(* CoDeSys 2.3.9.59 project: PD4.pro *)
(* Libraries: Standard.lib, SYSLIBCALLBACK.LIB *)

(* PLC configuration (modules and I/O channels)
Configuration EC4P-200 [Root] node -1, in %IB0 out %QB0 {EC4P_RestartPwrOn = WARMSTART; EC4P_MaxCycleTime = 20; EC4P_Com1BaudRate = 38400; EC4P_CAN1BaudRate = 125KBaud; EC4P_RoutingId = 127; EC4P_EasyNetId = 1; EC4P_EasyNetCfg = 0; EC4P_EasyNetCycleTime = 50; EC4P_RoutingChannel = CAN1; EC4P_IPFlags = 0; EC4P_IPAddress = 0; EC4P_SubNetMask = 0; EC4P_DefaultGateway = 0; EC4P_SummerWinterFlags = 0; EC4P_SummerWinterRule1 = 0; EC4P_SummerWinterRule2 = 0}
  Local I/O [EC4P_LocalIO] node 0, in %IB0 out %QB0 {EC4P_LocalInt = 0}
    I1 AT %IX0.0 [LocalBitInput] Input I1
    I2 AT %IX0.1 [LocalBitInput] Input I2
    I3 AT %IX0.2 [LocalBitInput] Input I3
    I4 AT %IX0.3 [LocalBitInput] Input I4
    I5 AT %IX0.4 [LocalBitInput] Input I5
    I6 AT %IX0.5 [LocalBitInput] Input I6
    I7 AT %IX0.6 [LocalBitInput] Input I7
    I8 AT %IX0.7 [LocalBitInput] Input I8
    I9 AT %IX1.0 [LocalBitInput] Input I9
    I10 AT %IX1.1 [LocalBitInput] Input I10
    I11 AT %IX1.2 [LocalBitInput] Input I11
    I12 AT %IX1.3 [LocalBitInput] Input I12
    I13 AT %IX1.4 [LocalDiagInput] Diagnostic Input I13
    I14 AT %IX1.5 [LocalDiagInput] Diagnostic Input I14
    I15 AT %IX1.6 [LocalDiagInput] Diagnostic Input I15
    I16 AT %IX1.7 [LocalDiagInput] Diagnostic Input I16
    I7_Analog AT %IW2 [LocalAnalogIn] Input I7, 10Bit, 0-10VDC
    I8_Analog AT %IW4 [LocalAnalogIn] Input I8, 10Bit, 0-10VDC
    I11_Analog AT %IW6 [LocalAnalogIn] Input I11, 10Bit, 0-10VDC
    I12_Analog AT %IW8 [LocalAnalogIn] Input I12, 10Bit, 0-10VDC
    Transistor Outputs [EC4P_TOutputs] node 0, in %IB10 out %QB0
      Q1 AT %QX0.0 [LocalBitOutput] Transistor-Output Q1
      Q2 AT %QX0.1 [LocalBitOutput] Transistor-Output Q2
      Q3 AT %QX0.2 [LocalBitOutput] Transistor-Output Q3
      Q4 AT %QX0.3 [LocalBitOutput] Transistor-Output Q4
      Q5 AT %QX0.4 [LocalBitOutput] Transistor-Output Q5
      Q6 AT %QX0.5 [LocalBitOutput] Transistor-Output Q6
      Q7 AT %QX0.6 [LocalBitOutput] Transistor-Output Q7
      Q8 AT %QX0.7 [LocalBitOutput] Transistor-Output Q8
    No Analog Output [EC4P_NoAnalogOutput] node 1, in %IB10 out %QB1
    No Keys [EC4P_NoKeys] node 2, in %IB10 out %QB1
    No Counter [EC4P_NoCounter] node 3, in %IB10 out %QB1
  Extension [EC4P_Extension] node 1, in %IB10 out %QB1
    No Extension [EC4P_NoExtension] node 0, in %IB10 out %QB1
*)

(* POU PLC_PRG, FBD *)
PROGRAM PLC_PRG
VAR
	sum: input_sum;
	segment: segment_driver;
END_VAR
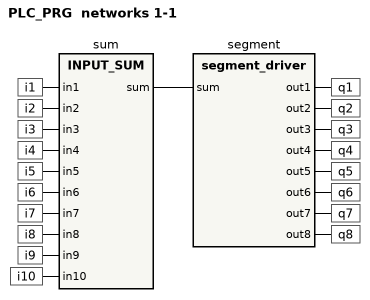
_FBD_ (* Function Block Diagram *)
NETWORK 1
	segment:segment_driver(sum: sum:INPUT_SUM(in1: i1, in2: i2, in3: i3, in4: i4, in5: i5, in6: i6, in7: i7, in8: i8, in9: i9, in10: i10), out2 => q2, out3 => q3, out4 => q4, out5 => q5, out6 => q6, out7 => q7, out8 => q8) => q1
_END_FBD_
(* the same logic as Structured Text *)
(* Network 1 *)
sum(in1 := i1, in2 := i2, in3 := i3, in4 := i4, in5 := i5, in6 := i6, in7 := i7, in8 := i8, in9 := i9, in10 := i10);
segment(sum := sum.sum);
q2 := segment.out2;
q3 := segment.out3;
q4 := segment.out4;
q5 := segment.out5;
q6 := segment.out6;
q7 := segment.out7;
q8 := segment.out8;
q1 := segment.out1;
END_PROGRAM

(* POU input_sum, ST *)
FUNCTION_BLOCK input_sum
VAR_INPUT
	in1, in2, in3, in4, in5, in6, in7, in8, in9, in10: BOOL;
END_VAR
VAR_OUTPUT
	sum: WORD;
END_VAR
VAR
END_VAR
sum := BOOL_TO_INT(in1) + BOOL_TO_INT(in2) + BOOL_TO_INT(in3) + BOOL_TO_INT(in4) + BOOL_TO_INT(in5) + BOOL_TO_INT(in6)+ BOOL_TO_INT(in7) + BOOL_TO_INT(in8) + BOOL_TO_INT(in9) + BOOL_TO_INT(in10);
END_FUNCTION_BLOCK

(* POU segment_driver, ST *)
FUNCTION_BLOCK segment_driver
VAR_INPUT
	sum: WORD;
END_VAR
VAR_OUTPUT
	out1, out2, out3, out4, out5, out6, out7, out8: BOOL;
END_VAR
VAR
END_VAR
CASE sum OF
0:
	out1 := 0;
	out2 := 0;
	out3 := 0;
	out4 := 0;
	out5 := 0;
	out6 := 0;
	out7 := 0;
	out8 := 1;
1:
	out1 := 0;
	out2 := 1;
	out3 := 0;
	out4 := 1;
	out5 := 1;
	out6 := 1;
	out7 := 1;
	out8 := 0;
2:
	out1 := 0;
	out2 := 0;
	out3 := 0;
	out4 := 1;
	out5 := 1;
	out6 := 0;
	out7 := 0;
	out8 := 0;
3:
	out1 := 1 ;
	out2 := 0;
	out3 := 1;
	out4 := 1;
	out5 := 1;
	out6 := 0;
	out7 := 1;
	out8 := 0;
4:
	out1 := 1;
	out2 := 1;
	out3 := 0;
	out4 := 1;
	out5 := 1;
	out6 := 0;
	out7 := 1;
	out8 := 0;
5:
	out1 := 1;
	out2 := 0;
	out3 := 1;
	out4 := 1;
	out5 := 1;
	out6 := 0;
	out7 := 1;
	out8 := 0;
6:
	out1 := 0;
	out2 := 1;
	out3 := 0;
	out4 := 0;
	out5 := 1;
	out6 := 0;
	out7 := 0;
	out8 := 0;
7:
	out1 := 0;
	out2 := 0;
	out3 := 0;
	out4 := 1;
	out5 := 1;
	out6 := 1;
	out7 := 0;
	out8 := 0;
8:
	out1 := 1;
	out2 := 1;
	out3 := 0;
	out4 := 1;
	out5 := 0;
	out6 := 1;
	out7 := 1;
	out8 := 0;
9:
	out1 := 1;
	out2 := 1;
	out3 := 0;
	out4 := 1;
	out5 := 1;
	out6 := 1;
	out7 := 0;
	out8 := 0;
10:
	out1 := 1;
	out2 := 1;
	out3 := 1;
	out4 := 1;
	out5 := 1;
	out6 := 1;
	out7 := 0;
	out8 := 0;
ELSE
	out1 := 0;
	out2 := 0;
	out3 := 0;
	out4 := 0;
	out5 := 0;
	out6 := 0;
	out7 := 0;
	out8 := 0;
END_CASE;
END_FUNCTION_BLOCK

(* Visualisation gui
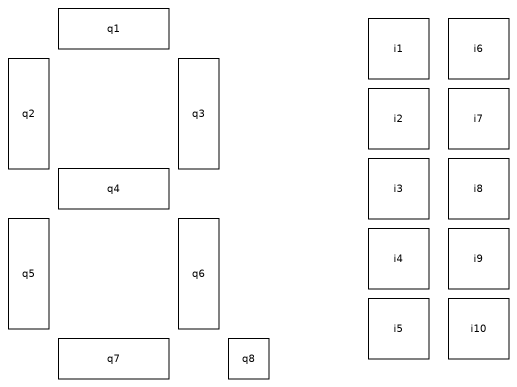
rectangle at (400,50)-(461,111): text "i1"; alarm colour if i1; toggles i1
rectangle at (400,120)-(461,181): text "i2"; alarm colour if i2; toggles i2
rectangle at (400,190)-(461,251): text "i3"; alarm colour if i3; toggles i3
rectangle at (480,50)-(541,111): text "i6"; alarm colour if i6; toggles i6
rectangle at (480,120)-(541,181): text "i7"; alarm colour if i7; toggles i7
rectangle at (480,190)-(541,251): text "i8"; alarm colour if i8; toggles i8
rectangle at (400,260)-(461,321): text "i4"; alarm colour if i4; toggles i4
rectangle at (400,330)-(461,391): text "i5"; alarm colour if i5; toggles i5
rectangle at (480,260)-(541,321): text "i9"; alarm colour if i9; toggles i9
rectangle at (480,330)-(541,391): text "i10"; alarm colour if i10; toggles i10
rectangle at (90,40)-(201,81): text "q1"; alarm colour if q1; toggles q1
rectangle at (40,90)-(81,201): text "q2"; alarm colour if q2; toggles q2
rectangle at (210,90)-(251,201): text "q3"; alarm colour if q3; toggles q3
rectangle at (90,200)-(201,241): text "q4"; alarm colour if q4; toggles q4
rectangle at (40,250)-(81,361): text "q5"; alarm colour if q5; toggles q5
rectangle at (210,250)-(251,361): text "q6"; alarm colour if q6; toggles q6
rectangle at (90,370)-(201,411): text "q7"; alarm colour if q7; toggles q7
rectangle at (260,370)-(301,411): text "q8"; alarm colour if q8; toggles q8
*)
